Universal Robots PolyScope program: Programa_2_ExternalControl.urp

Program Programa_2_ExternalControl (createdIn=3.15.8.106339 lastSavedIn=3.15.8.106339 directory=/ursim/programs installation=practica_simulacion robotSerialNumber=2018359999)
Calibrated DH parameters: a=[0, -0.425, -0.39225, 0, 0, 0]; d=[0.089159, 0, 0, 0.10915, 0.09465, 0.0823]; alpha=[1.570796, 0, 0, 1.570796, -1.570796, 0]; deltaTheta=[0, 0, 0, 0, 0, 0]
Robot Program (runOnlyOnce=true motionType=MoveJ speed=0.4 acceleration=0.6 useActiveTCP=true)
  'SOLO URSim — Brayan Mateo Bravo Losada'
  Script file /ursim/programs/Programa_2_ExternalControl_rutina.script
    | sim = rpc_factory("xmlrpc", "http://172.17.0.1:40404/RPC2")
    | set_standard_digital_out(0, True)
    | sim.event("salida_control_alta", get_actual_tcp_pose())
    | popup("El control se compartira con ROS 2 simulado 5 segundos despues de confirmar.", title="Programa 2", blocking=True)
    | sim.event("popup_control_confirmado", get_actual_tcp_pose())
    | sleep(5.0)
    | sim.event("espera_5s_terminada", get_actual_tcp_pose())
  URCap External Control (External Control, FZI Research Center for Information Technology)
  Script file /ursim/programs/Programa_2_devolver.script
    | set_standard_digital_out(0, False)
    | sim.event("control_devuelto", get_actual_tcp_pose())
